// TIA Portal V18 export
// export: Created 2025-12-01T17:51:20.5638131Z, ExportSetting None, DisplayName Totally Integrated Automation Portal, DisplayVersion V18 Update 5, DisplayName TIA Portal Openness, DisplayVersion V18 Update 5, DisplayName TIA Portal Teamcenter Gateway, DisplayVersion V18, DisplayName TIA Portal Version Control Interface, DisplayVersion V18, DisplayName STEP 7 Professional, DisplayVersion V18 Update 5, DisplayName STEP 7 Safety, DisplayVersion V18, DisplayName WinCC Professional, DisplayVersion V18 Update 5
DATA_BLOCK "MotorContro_DB_11"   // DB3111
// stored: AutoNumber false, InstanceOfName MotorContro, InstanceOfType FB
"MotorContro"
   // VAR_INPUT
   //    iAlwaysTrue : Bool;
   //    iSysRun : Bool;
   //    iReset : Bool;
   //    iAuto : Bool;
   //    iManual : Bool;
   //    i_ParySensor : Bool;
   //    i_Alarm : Bool;
   //    iType : Int;
   //    i_RunInTimeDelay : Time;
   //    i_RunOutTimeDelay : Time;
   //    i_Interlock : Bool;
   // END_VAR
   // VAR_IN_OUT
   //    Control : "Motor_Control";
   // END_VAR
   // VAR
   //    TON : Array[0..5] of TON_TIME;
   //    Zero { S7_SetPoint := 'True'} : Array[0..15] of Bool;
   // END_VAR
BEGIN
END_DATA_BLOCK
